(* PLC project Unnamed, Unknown Unnamed 1 *)
(* stored: creationDateTime 2025-05-15T16:41:17, modificationDateTime 2025-05-15T17:50:37 *)

PROGRAM waterESP
  VAR
    pulse : BOOL;
  END_VAR
  VAR
    counter_enable AT %QX0.0 : BOOL;
    counter_reset AT %QX0.1 : BOOL;
    counter_q AT %QX0.2 : BOOL;
    counter_max AT %QW0 : INT := 10;
  END_VAR
  VAR
    CTU0 : CTU;
    counter_value : INT;
    TON1 : TON;
    TOF0 : TOF;
  END_VAR
  VAR  (* added by the conversion: wires and edge detectors of the diagram *)
    R_TRIG1 : R_TRIG;
  END_VAR

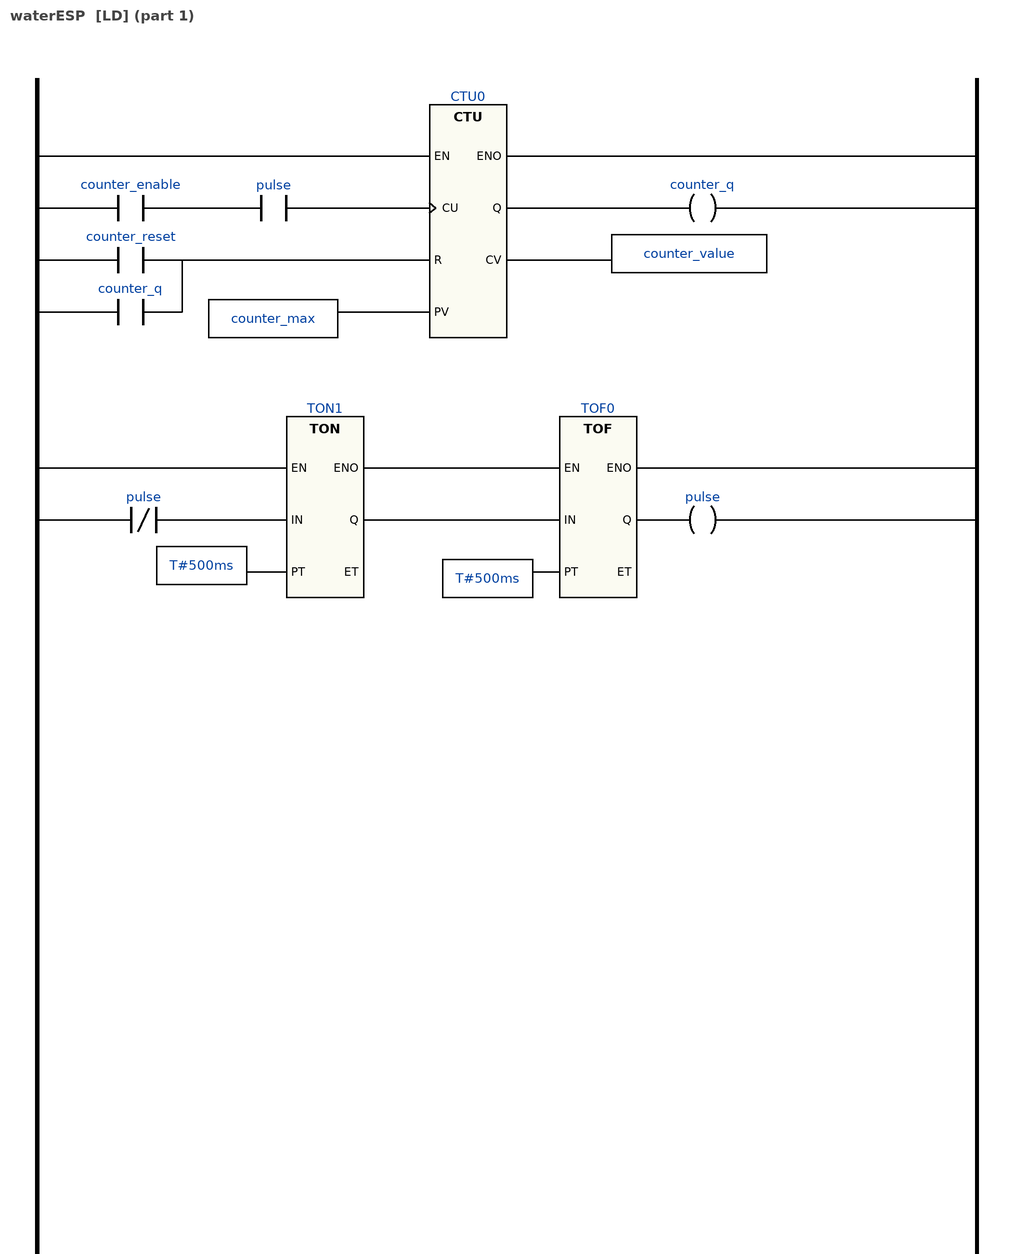
(* LD diagram, written out as Structured Text *)
R_TRIG1(CLK := counter_enable AND pulse);
CTU0(CU := R_TRIG1.Q, R := counter_reset OR counter_q, PV := counter_max);
counter_value := CTU0.CV;
counter_q := CTU0.Q;
TON1(IN := NOT pulse, PT := T#500ms);
TOF0(EN := TON1.ENO, IN := TON1.Q, PT := T#500ms);
pulse := TOF0.Q;
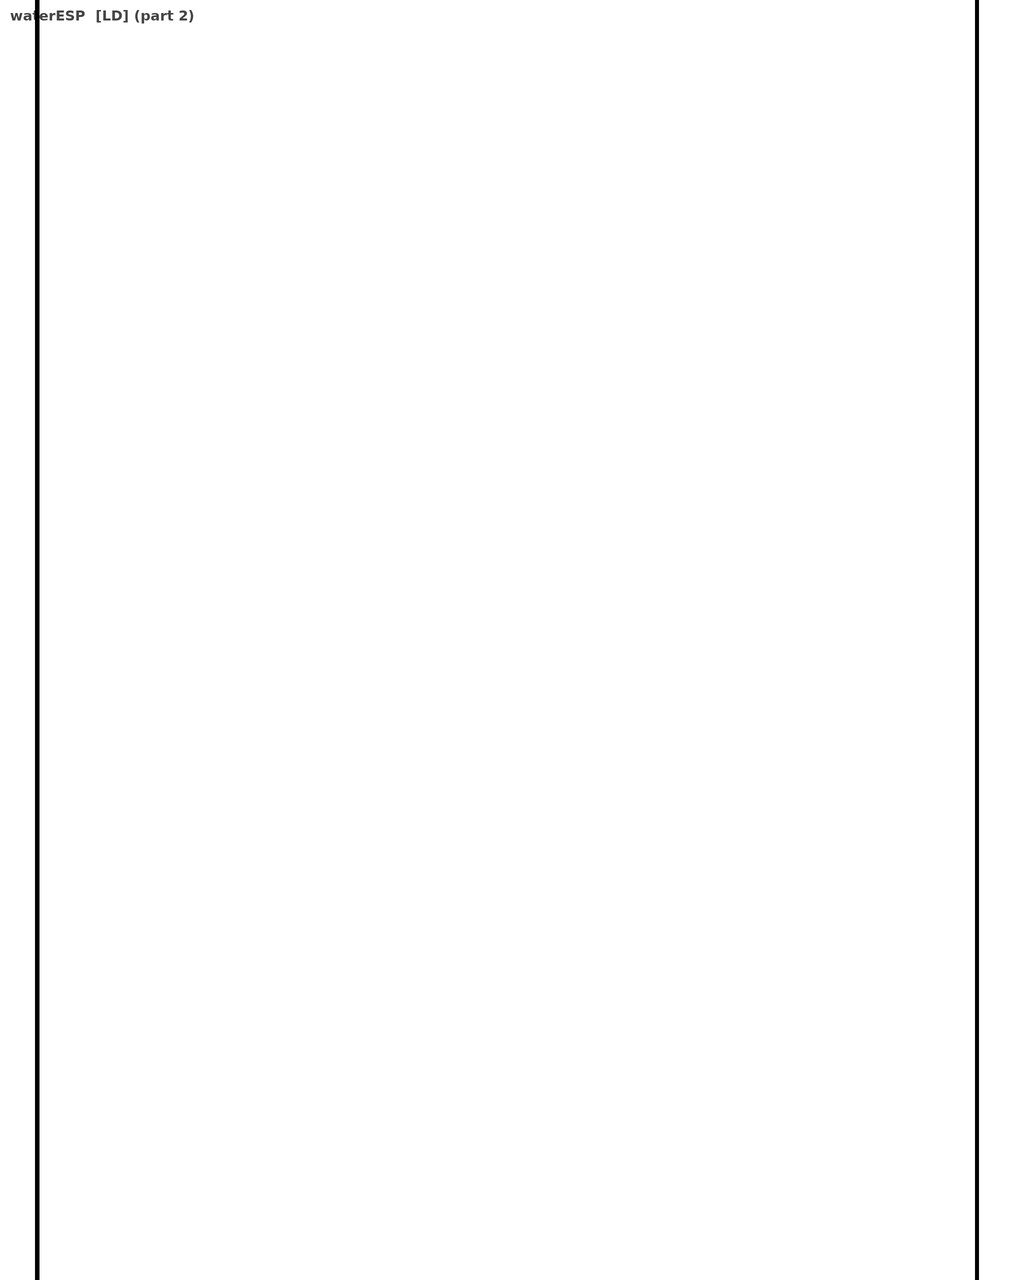
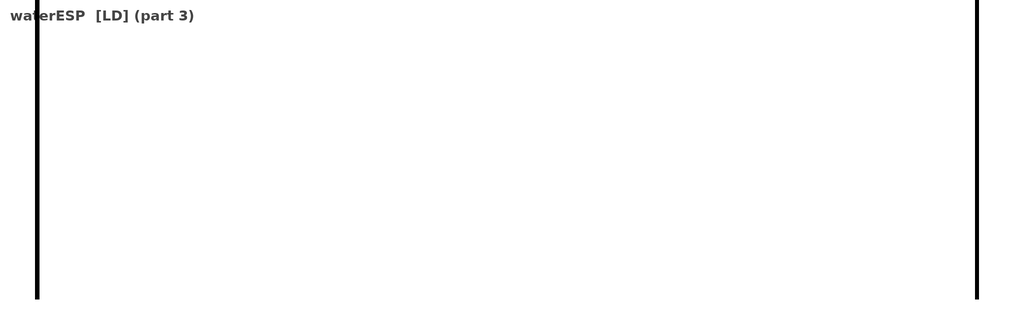
END_PROGRAM

CONFIGURATION Config0
  RESOURCE Res0 ON PLC
    TASK task0(INTERVAL := T#20ms, PRIORITY := 0);
    PROGRAM instance0 WITH task0 : waterESP;
  END_RESOURCE
END_CONFIGURATION
